// TIA Portal V15.1 program export: 0 tag tables, 0 data types, 0 data blocks, 4 code blocks (in call order from the OBs), 1 instance data blocks

ORGANIZATION_BLOCK "Main"   // OB1, LAD, ProgramCycle
TITLE = "Main Program Sweep (Cycle)"
{ S7_Optimized_Access := 'TRUE' }
VERSION : 0.1
// stored: AutoNumber true, CodeModifiedDate 2022-03-08T11:13:54.5164113Z, CompileDate 2022-03-08T11:13:55.9851651Z, ConstantName OB_Main, CreationDate 2022-02-28T09:16:09.6965758Z, EventClass Program cycle, HandleErrorsWithinBlock false, InterfaceModifiedDate 2022-02-28T09:18:02.6969839Z, IsConsistent true, IsIECCheckEnabled false, IsKnowHowProtected false, IsWriteProtected false, ModifiedDate 2022-03-08T11:13:54.5164113Z, ParameterModified 2022-02-28T09:18:02.6969839Z, PLCSimAdvancedSupport false, PriorityNumber 1, ProcessImagePartNumber 65535, SetENOAutomatically False, StructureModified 2022-02-28T09:18:02.6969839Z
   VAR_INPUT
      Initial_Call : Bool;   // Initial call of this OB
      Remanence : Bool;   // =True, if remanent data are available
   END_VAR
BEGIN

REGION Network 1
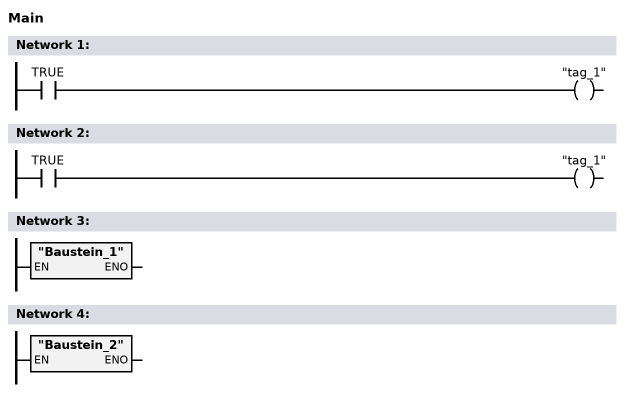
   RUNG wire#powerrail
      Contact( TRUE )
      Coil( "tag_1" )
   END_RUNG
   // the same network as SCL:
   "tag_1" := TRUE;
END_REGION

REGION Network 2
   RUNG wire#powerrail
      Contact( TRUE )
      Coil( "tag_1" )
   END_RUNG
   // the same network as SCL:
   "tag_1" := TRUE;
END_REGION

REGION Network 3
   RUNG wire#powerrail
      "Baustein_1"()
   END_RUNG
   // the same network as SCL:
   "Baustein_1"();
END_REGION

REGION Network 4
   RUNG wire#powerrail
      "Baustein_2"()
   END_RUNG
   // the same network as SCL:
   "Baustein_2"();
END_REGION
END_ORGANIZATION_BLOCK

FUNCTION "Baustein_1" : Void   // FC1, LAD
{ S7_Optimized_Access := 'TRUE' }
VERSION : 0.1
// stored: AutoNumber true, CodeModifiedDate 2022-03-08T11:13:52.6713816Z, CompileDate 2022-03-08T11:13:55.9071944Z, CreationDate 2022-03-08T11:10:18.1755096Z, HandleErrorsWithinBlock false, InterfaceModifiedDate 2022-03-08T11:10:18.1755096Z, IsConsistent true, IsIECCheckEnabled false, IsKnowHowProtected false, IsWriteProtected false, LibraryConformanceStatus Fehler: Der Baustein enthält Aufrufe von Einzelinstanzen. Warnung: Der Baustein enthält direkte Zugriffe auf Eingänge, Ausgänge, Merker, indirekte Zugriffe auf Register oder indirekte Zugriffe auf externe, zum Übersetzungszeitpunkt unbekannte Speicherbereiche., ModifiedDate 2022-03-08T11:13:52.6713816Z, ParameterModified 2022-03-08T11:10:18.1755096Z, PLCSimAdvancedSupport false, SetENOAutomatically False, StructureModified 2022-03-08T11:10:18.1755096Z, UDAEnableTagReadback false
BEGIN

REGION Network 1
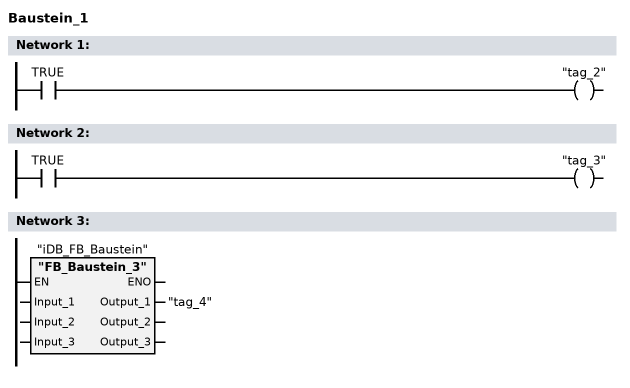
   RUNG wire#powerrail
      Contact( TRUE )
      Coil( "tag_2" )
   END_RUNG
   // the same network as SCL:
   "tag_2" := TRUE;
END_REGION

REGION Network 2
   RUNG wire#powerrail
      Contact( TRUE )
      Coil( "tag_3" )
   END_RUNG
   // the same network as SCL:
   "tag_3" := TRUE;
END_REGION

REGION Network 3
   RUNG wire#powerrail
      "iDB_FB_Baustein"(Input_1 :=, Input_2 :=, Input_3 :=, Output_1 => "tag_4", Output_2 =>, Output_3 =>)
   END_RUNG
   // the same network as SCL:
   "iDB_FB_Baustein"(Output_1 => "tag_4");   // "FB_Baustein_3"
END_REGION
END_FUNCTION

FUNCTION_BLOCK "FB_Baustein_3"   // FB1, SCL
{ S7_Optimized_Access := 'TRUE' }
VERSION : 0.1
// stored: AutoNumber true, CodeModifiedDate 2022-03-08T11:13:52.8896608Z, CompileDate 2022-03-08T11:13:54.0933934Z, CreationDate 2022-03-08T11:12:33.2792339Z, DownloadWithoutReinit false, HandleErrorsWithinBlock false, InterfaceModifiedDate 2022-03-08T11:12:52.1304591Z, IsConsistent true, IsIECCheckEnabled false, IsKnowHowProtected false, ISMultiInstanceCapable true, IsRetainMemResEnabled false, IsWriteProtected false, LibraryConformanceStatus Das Objekt ist bibliothekskonform., MemoryReserve 100, ModifiedDate 2022-03-08T11:13:53.4529134Z, ParameterModified 2022-03-08T11:12:52.1304591Z, PLCSimAdvancedSupport false, SetENOAutomatically False, StructureModified 2022-03-08T11:12:52.1304591Z, UDAEnableTagReadback false
   VAR_INPUT
      Input_1 : Bool;
      Input_2 : Bool;
      Input_3 : Bool;
   END_VAR
   VAR_OUTPUT
      Output_1 : Bool;
      Output_2 : Bool;
      Output_3 : Bool;
   END_VAR
BEGIN
END_FUNCTION_BLOCK

FUNCTION "Baustein_2" : Void   // FC2, LAD
{ S7_Optimized_Access := 'TRUE' }
VERSION : 0.1
// stored: AutoNumber true, CodeModifiedDate 2022-03-08T11:13:52.6871257Z, CompileDate 2022-03-08T11:13:55.7033463Z, CreationDate 2022-03-08T11:10:33.1505035Z, HandleErrorsWithinBlock false, InterfaceModifiedDate 2022-03-08T11:10:33.1505035Z, IsConsistent true, IsIECCheckEnabled false, IsKnowHowProtected false, IsWriteProtected false, LibraryConformanceStatus Fehler: Der Baustein enthält Aufrufe von Einzelinstanzen. Warnung: Der Baustein enthält direkte Zugriffe auf Eingänge, Ausgänge, Merker, indirekte Zugriffe auf Register oder indirekte Zugriffe auf externe, zum Übersetzungszeitpunkt unbekannte Speicherbereiche., ModifiedDate 2022-03-08T11:13:52.6871257Z, ParameterModified 2022-03-08T11:10:33.1505035Z, PLCSimAdvancedSupport false, SetENOAutomatically False, StructureModified 2022-03-08T11:10:33.1505035Z, UDAEnableTagReadback false
BEGIN

REGION Network 1
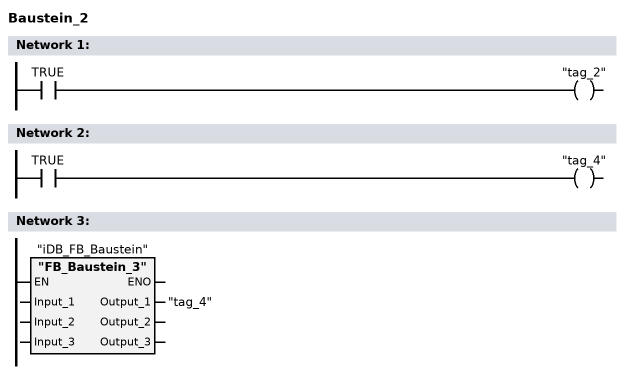
   RUNG wire#powerrail
      Contact( TRUE )
      Coil( "tag_2" )
   END_RUNG
   // the same network as SCL:
   "tag_2" := TRUE;
END_REGION

REGION Network 2
   RUNG wire#powerrail
      Contact( TRUE )
      Coil( "tag_4" )
   END_RUNG
   // the same network as SCL:
   "tag_4" := TRUE;
END_REGION

REGION Network 3
   RUNG wire#powerrail
      "iDB_FB_Baustein"(Input_1 :=, Input_2 :=, Input_3 :=, Output_1 => "tag_4", Output_2 =>, Output_3 =>)
   END_RUNG
   // the same network as SCL:
   "iDB_FB_Baustein"(Output_1 => "tag_4");   // "FB_Baustein_3"
END_REGION
END_FUNCTION

DATA_BLOCK "iDB_FB_Baustein"   // DB1
{ S7_Optimized_Access := 'TRUE' }
VERSION : 0.1
// stored: AutoNumber true, CodeModifiedDate 2022-03-08T11:13:20.8295301Z, CompileDate 2022-03-08T11:13:54.4692283Z, CreationDate 2022-03-08T11:13:20.5332262Z, DBAccessibleFromOPCUA true, DownloadWithoutReinit false, InstanceOfName FB_Baustein_3, InstanceOfNumber 1, InstanceOfType FB, InterfaceModifiedDate 2022-03-08T11:12:52.1304591Z, IsConsistent true, IsKnowHowProtected false, IsRetainMemResEnabled false, MemoryReserve 100, ModifiedDate 2022-03-08T11:13:20.8295301Z, ParameterModified 2022-03-08T11:12:52.1304591Z, StructureModified 2022-03-08T11:12:52.1304591Z, UDAEnableTagReadback false
"FB_Baustein_3"
BEGIN
END_DATA_BLOCK
